SUBAPPLICATION Uebung_020d_AX (* DigitalInput_I1 auf DigitalOutput_Q1; TOF Ausschaltverzögert; aufgelöst *)
  (* Standard: 61499-2; Description: Copyright (c) 2023 Meisterschulen am Ostbahnhof This program and the accompanying materials are made available under the terms of the Eclipse Public License 2.0 which is available at https://www.eclipse.org/legal/epl-2.0/ SPDX-License-Identifier: EPL-2.0 *)
  (* Version 1.0, 2026-01-16, Franz Höpfinger, Meisterschulen am Ostbahnhof, initial API and implementation and/or initial documentation *)
  PACKAGE Uebungen;
  IMPORT logiBUS::io::DI::logiBUS_DI::Input_I1;
  IMPORT logiBUS::io::DQ::logiBUS_DO::Output_Q1;
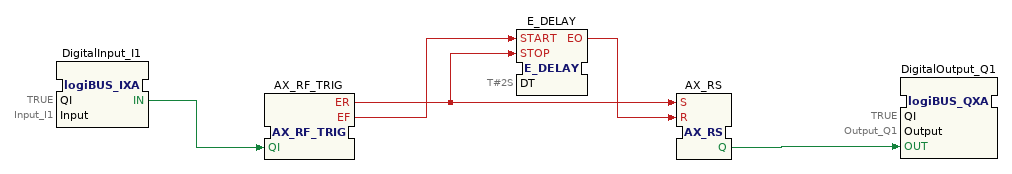
  FBS
    DigitalInput_I1 : logiBUS::io::DI::logiBUS_IXA(QI := TRUE, Input := Input_I1);
    AX_RF_TRIG : adapter::events::unidirectional::AX_RF_TRIG;
    AX_RS : adapter::events::unidirectional::AX_RS;
    E_DELAY : iec61499::events::E_DELAY(DT := T#2S);
    DigitalOutput_Q1 : logiBUS::io::DQ::logiBUS_QXA(QI := TRUE, Output := Output_Q1);
  END_FBS
  EVENT_CONNECTIONS
    AX_RF_TRIG.ER TO AX_RS.S;
    AX_RF_TRIG.EF TO E_DELAY.START;
    E_DELAY.EO TO AX_RS.R;
    AX_RF_TRIG.ER TO E_DELAY.STOP;
  END_CONNECTIONS
  ADAPTER_CONNECTIONS
    DigitalInput_I1.IN TO AX_RF_TRIG.QI;
    AX_RS.Q TO DigitalOutput_Q1.OUT;
  END_CONNECTIONS
END_SUBAPPLICATION
